// TIA Portal V19 export
DATA_BLOCK "MwFakCalc_PERS"   // DB132
// stored: MemoryReserve 100
   VAR RETAIN
      PersistentValues : "udt_MwFacCalc_Pers";
   END_VAR
BEGIN
   PersistentValues.Data.MaterialPresence := TRUE;
   PersistentValues.Data.Reg[1].ID := 713;
   PersistentValues.Data.Reg[2].ID := 712;
   PersistentValues.Data.Reg[3].ID := 711;
   PersistentValues.Data.Reg[4].ID := 710;
   PersistentValues.Data.Reg[5].ID := 709;
   PersistentValues.Data.Reg[6].ID := 708;
   PersistentValues.Data.Reg[7].ID := 707;
   PersistentValues.Data.Reg[8].ID := 706;
   PersistentValues.Data.Reg[9].ID := 705;
   PersistentValues.Data.Reg[10].ID := 704;
   PersistentValues.Data.Reg[1].FAK := 1.00032760149922;
   PersistentValues.Data.Reg[2].FAK := 1.00025286183891;
   PersistentValues.Data.Reg[3].FAK := 1.00034141784116;
   PersistentValues.Data.Reg[4].FAK := 1.00032858034714;
   PersistentValues.Data.Reg[5].FAK := 1.00027275466515;
   PersistentValues.Data.Reg[6].FAK := 1.00033876404002;
   PersistentValues.Data.Reg[7].FAK := 1.00043144089834;
   PersistentValues.Data.Reg[8].FAK := 1.00027468282716;
   PersistentValues.Data.Reg[9].FAK := 1.0002702312408;
   PersistentValues.Data.Reg[10].FAK := 1.00040598281433;
   PersistentValues.Data.Reg[1].FAK_PS := 1.00033187802923;
   PersistentValues.Data.Reg[2].FAK_PS := 1.0002428384096;
   PersistentValues.Data.Reg[3].FAK_PS := 1.00034713591431;
   PersistentValues.Data.Reg[4].FAK_PS := 1.0003300372471;
   PersistentValues.Data.Reg[5].FAK_PS := 1.00028276221556;
   PersistentValues.Data.Reg[6].FAK_PS := 1.0003416145074;
   PersistentValues.Data.Reg[7].FAK_PS := 1.00041568993821;
   PersistentValues.Data.Reg[8].FAK_PS := 1.00027756475559;
   PersistentValues.Data.Reg[9].FAK_PS := 1.00025879029114;
   PersistentValues.Data.Reg[10].FAK_PS := 1.00039311435194;
   PersistentValues.Data.Reg[1].TP_W_Meas1Reg.ID := 1347;
   PersistentValues.Data.Reg[2].TP_W_Meas1Reg.ID := 1345;
   PersistentValues.Data.Reg[3].TP_W_Meas1Reg.ID := 1343;
   PersistentValues.Data.Reg[4].TP_W_Meas1Reg.ID := 1341;
   PersistentValues.Data.Reg[5].TP_W_Meas1Reg.ID := 1339;
   PersistentValues.Data.Reg[6].TP_W_Meas1Reg.ID := 1337;
   PersistentValues.Data.Reg[7].TP_W_Meas1Reg.ID := 1335;
   PersistentValues.Data.Reg[8].TP_W_Meas1Reg.ID := 1333;
   PersistentValues.Data.Reg[9].TP_W_Meas1Reg.ID := 1331;
   PersistentValues.Data.Reg[10].TP_W_Meas1Reg.ID := 1329;
   PersistentValues.Data.Reg[1].TP_W_Meas1Reg.Position := 900953.878;
   PersistentValues.Data.Reg[2].TP_W_Meas1Reg.Position := 898853.79;
   PersistentValues.Data.Reg[3].TP_W_Meas1Reg.Position := 896756.481;
   PersistentValues.Data.Reg[4].TP_W_Meas1Reg.Position := 895002.073;
   PersistentValues.Data.Reg[5].TP_W_Meas1Reg.Position := 892900.793;
   PersistentValues.Data.Reg[6].TP_W_Meas1Reg.Position := 890799.166;
   PersistentValues.Data.Reg[7].TP_W_Meas1Reg.Position := 888692.332;
   PersistentValues.Data.Reg[8].TP_W_Meas1Reg.Position := 886941.647;
   PersistentValues.Data.Reg[9].TP_W_Meas1Reg.Position := 884838.939;
   PersistentValues.Data.Reg[10].TP_W_Meas1Reg.Position := 882730.285;
   PersistentValues.Data.Reg[1].TP_G_Meas1Reg.ID := 1346;
   PersistentValues.Data.Reg[2].TP_G_Meas1Reg.ID := 1344;
   PersistentValues.Data.Reg[3].TP_G_Meas1Reg.ID := 1342;
   PersistentValues.Data.Reg[4].TP_G_Meas1Reg.ID := 1340;
   PersistentValues.Data.Reg[5].TP_G_Meas1Reg.ID := 1338;
   PersistentValues.Data.Reg[6].TP_G_Meas1Reg.ID := 1336;
   PersistentValues.Data.Reg[7].TP_G_Meas1Reg.ID := 1334;
   PersistentValues.Data.Reg[8].TP_G_Meas1Reg.ID := 1332;
   PersistentValues.Data.Reg[9].TP_G_Meas1Reg.ID := 1330;
   PersistentValues.Data.Reg[10].TP_G_Meas1Reg.ID := 1328;
   PersistentValues.Data.Reg[1].TP_G_Meas1Reg.Position := -650.875;
   PersistentValues.Data.Reg[2].TP_G_Meas1Reg.Position := -651.608;
   PersistentValues.Data.Reg[3].TP_G_Meas1Reg.Position := -652.018;
   PersistentValues.Data.Reg[4].TP_G_Meas1Reg.Position := -651.902;
   PersistentValues.Data.Reg[5].TP_G_Meas1Reg.Position := -652.251;
   PersistentValues.Data.Reg[6].TP_G_Meas1Reg.Position := -651.557;
   PersistentValues.Data.Reg[7].TP_G_Meas1Reg.Position := -651.833;
   PersistentValues.Data.Reg[8].TP_G_Meas1Reg.Position := -650.823;
   PersistentValues.Data.Reg[9].TP_G_Meas1Reg.Position := -651.386;
   PersistentValues.Data.Reg[10].TP_G_Meas1Reg.Position := -652.001;
   PersistentValues.Data.Reg[1].TP_W_Meas2Reg.ID := 1348;
   PersistentValues.Data.Reg[2].TP_W_Meas2Reg.ID := 1346;
   PersistentValues.Data.Reg[3].TP_W_Meas2Reg.ID := 1344;
   PersistentValues.Data.Reg[4].TP_W_Meas2Reg.ID := 1342;
   PersistentValues.Data.Reg[5].TP_W_Meas2Reg.ID := 1340;
   PersistentValues.Data.Reg[6].TP_W_Meas2Reg.ID := 1338;
   PersistentValues.Data.Reg[7].TP_W_Meas2Reg.ID := 1336;
   PersistentValues.Data.Reg[8].TP_W_Meas2Reg.ID := 1334;
   PersistentValues.Data.Reg[9].TP_W_Meas2Reg.ID := 1332;
   PersistentValues.Data.Reg[10].TP_W_Meas2Reg.ID := 1330;
   PersistentValues.Data.Reg[1].TP_W_Meas2Reg.Position := 901652.898;
   PersistentValues.Data.Reg[2].TP_W_Meas2Reg.Position := 899553.777;
   PersistentValues.Data.Reg[3].TP_W_Meas2Reg.Position := 897456.503;
   PersistentValues.Data.Reg[4].TP_W_Meas2Reg.Position := 895702.054;
   PersistentValues.Data.Reg[5].TP_W_Meas2Reg.Position := 893601.056;
   PersistentValues.Data.Reg[6].TP_W_Meas2Reg.Position := 891498.768;
   PersistentValues.Data.Reg[7].TP_W_Meas2Reg.Position := 889392.312;
   PersistentValues.Data.Reg[8].TP_W_Meas2Reg.Position := 887640.635;
   PersistentValues.Data.Reg[9].TP_W_Meas2Reg.Position := 885538.34;
   PersistentValues.Data.Reg[10].TP_W_Meas2Reg.Position := 883429.822;
   PersistentValues.Data.Reg[1].TP_G_Meas2Reg.ID := 1347;
   PersistentValues.Data.Reg[2].TP_G_Meas2Reg.ID := 1345;
   PersistentValues.Data.Reg[3].TP_G_Meas2Reg.ID := 1343;
   PersistentValues.Data.Reg[4].TP_G_Meas2Reg.ID := 1341;
   PersistentValues.Data.Reg[5].TP_G_Meas2Reg.ID := 1339;
   PersistentValues.Data.Reg[6].TP_G_Meas2Reg.ID := 1337;
   PersistentValues.Data.Reg[7].TP_G_Meas2Reg.ID := 1335;
   PersistentValues.Data.Reg[8].TP_G_Meas2Reg.ID := 1333;
   PersistentValues.Data.Reg[9].TP_G_Meas2Reg.ID := 1331;
   PersistentValues.Data.Reg[10].TP_G_Meas2Reg.ID := 1329;
   PersistentValues.Data.Reg[1].TP_G_Meas2Reg.Position := 48.374;
   PersistentValues.Data.Reg[2].TP_G_Meas2Reg.Position := 48.556;
   PersistentValues.Data.Reg[3].TP_G_Meas2Reg.Position := 48.243;
   PersistentValues.Data.Reg[4].TP_G_Meas2Reg.Position := 48.309;
   PersistentValues.Data.Reg[5].TP_G_Meas2Reg.Position := 48.203;
   PersistentValues.Data.Reg[6].TP_G_Meas2Reg.Position := 48.282;
   PersistentValues.Data.Reg[7].TP_G_Meas2Reg.Position := 48.449;
   PersistentValues.Data.Reg[8].TP_G_Meas2Reg.Position := 48.357;
   PersistentValues.Data.Reg[9].TP_G_Meas2Reg.Position := 48.204;
   PersistentValues.Data.Reg[10].TP_G_Meas2Reg.Position := 47.82;
   PersistentValues.Data.Reg[1].PS_W_Meas1Reg.ID := 217;
   PersistentValues.Data.Reg[2].PS_W_Meas1Reg.ID := 215;
   PersistentValues.Data.Reg[3].PS_W_Meas1Reg.ID := 213;
   PersistentValues.Data.Reg[4].PS_W_Meas1Reg.ID := 211;
   PersistentValues.Data.Reg[5].PS_W_Meas1Reg.ID := 209;
   PersistentValues.Data.Reg[6].PS_W_Meas1Reg.ID := 207;
   PersistentValues.Data.Reg[7].PS_W_Meas1Reg.ID := 205;
   PersistentValues.Data.Reg[8].PS_W_Meas1Reg.ID := 203;
   PersistentValues.Data.Reg[9].PS_W_Meas1Reg.ID := 201;
   PersistentValues.Data.Reg[10].PS_W_Meas1Reg.ID := 199;
   PersistentValues.Data.Reg[1].PS_W_Meas1Reg.Position := 900953.482;
   PersistentValues.Data.Reg[2].PS_W_Meas1Reg.Position := 898853.373;
   PersistentValues.Data.Reg[3].PS_W_Meas1Reg.Position := 896756.134;
   PersistentValues.Data.Reg[4].PS_W_Meas1Reg.Position := 895001.723;
   PersistentValues.Data.Reg[5].PS_W_Meas1Reg.Position := 892900.467;
   PersistentValues.Data.Reg[6].PS_W_Meas1Reg.Position := 890798.798;
   PersistentValues.Data.Reg[7].PS_W_Meas1Reg.Position := 888691.934;
   PersistentValues.Data.Reg[8].PS_W_Meas1Reg.Position := 886941.298;
   PersistentValues.Data.Reg[9].PS_W_Meas1Reg.Position := 884838.507;
   PersistentValues.Data.Reg[10].PS_W_Meas1Reg.Position := 882729.938;
   PersistentValues.Data.Reg[1].PS_G_Meas1Reg.ID := 217;
   PersistentValues.Data.Reg[2].PS_G_Meas1Reg.ID := 215;
   PersistentValues.Data.Reg[3].PS_G_Meas1Reg.ID := 213;
   PersistentValues.Data.Reg[4].PS_G_Meas1Reg.ID := 211;
   PersistentValues.Data.Reg[5].PS_G_Meas1Reg.ID := 209;
   PersistentValues.Data.Reg[6].PS_G_Meas1Reg.ID := 207;
   PersistentValues.Data.Reg[7].PS_G_Meas1Reg.ID := 205;
   PersistentValues.Data.Reg[8].PS_G_Meas1Reg.ID := 203;
   PersistentValues.Data.Reg[9].PS_G_Meas1Reg.ID := 201;
   PersistentValues.Data.Reg[10].PS_G_Meas1Reg.ID := 199;
   PersistentValues.Data.Reg[1].PS_G_Meas1Reg.Position := -651.256;
   PersistentValues.Data.Reg[2].PS_G_Meas1Reg.Position := -652.0;
   PersistentValues.Data.Reg[3].PS_G_Meas1Reg.Position := -652.349;
   PersistentValues.Data.Reg[4].PS_G_Meas1Reg.Position := -652.229;
   PersistentValues.Data.Reg[5].PS_G_Meas1Reg.Position := -652.553;
   PersistentValues.Data.Reg[6].PS_G_Meas1Reg.Position := -651.902;
   PersistentValues.Data.Reg[7].PS_G_Meas1Reg.Position := -652.202;
   PersistentValues.Data.Reg[8].PS_G_Meas1Reg.Position := -651.153;
   PersistentValues.Data.Reg[9].PS_G_Meas1Reg.Position := -651.791;
   PersistentValues.Data.Reg[10].PS_G_Meas1Reg.Position := -652.328;
   PersistentValues.Data.Reg[1].PS_W_Meas2Reg.ID := 218;
   PersistentValues.Data.Reg[2].PS_W_Meas2Reg.ID := 216;
   PersistentValues.Data.Reg[3].PS_W_Meas2Reg.ID := 214;
   PersistentValues.Data.Reg[4].PS_W_Meas2Reg.ID := 212;
   PersistentValues.Data.Reg[5].PS_W_Meas2Reg.ID := 210;
   PersistentValues.Data.Reg[6].PS_W_Meas2Reg.ID := 208;
   PersistentValues.Data.Reg[7].PS_W_Meas2Reg.ID := 206;
   PersistentValues.Data.Reg[8].PS_W_Meas2Reg.ID := 204;
   PersistentValues.Data.Reg[9].PS_W_Meas2Reg.ID := 202;
   PersistentValues.Data.Reg[10].PS_W_Meas2Reg.ID := 200;
   PersistentValues.Data.Reg[1].PS_W_Meas2Reg.Position := 901652.534;
   PersistentValues.Data.Reg[2].PS_W_Meas2Reg.Position := 899553.427;
   PersistentValues.Data.Reg[3].PS_W_Meas2Reg.Position := 897456.148;
   PersistentValues.Data.Reg[4].PS_W_Meas2Reg.Position := 895701.644;
   PersistentValues.Data.Reg[5].PS_W_Meas2Reg.Position := 893600.702;
   PersistentValues.Data.Reg[6].PS_W_Meas2Reg.Position := 891498.417;
   PersistentValues.Data.Reg[7].PS_W_Meas2Reg.Position := 889391.975;
   PersistentValues.Data.Reg[8].PS_W_Meas2Reg.Position := 887640.234;
   PersistentValues.Data.Reg[9].PS_W_Meas2Reg.Position := 885537.915;
   PersistentValues.Data.Reg[10].PS_W_Meas2Reg.Position := 883429.48;
   PersistentValues.Data.Reg[1].PS_G_Meas2Reg.ID := 218;
   PersistentValues.Data.Reg[2].PS_G_Meas2Reg.ID := 216;
   PersistentValues.Data.Reg[3].PS_G_Meas2Reg.ID := 214;
   PersistentValues.Data.Reg[4].PS_G_Meas2Reg.ID := 212;
   PersistentValues.Data.Reg[5].PS_G_Meas2Reg.ID := 210;
   PersistentValues.Data.Reg[6].PS_G_Meas2Reg.ID := 208;
   PersistentValues.Data.Reg[7].PS_G_Meas2Reg.ID := 206;
   PersistentValues.Data.Reg[8].PS_G_Meas2Reg.ID := 204;
   PersistentValues.Data.Reg[9].PS_G_Meas2Reg.ID := 202;
   PersistentValues.Data.Reg[10].PS_G_Meas2Reg.ID := 200;
   PersistentValues.Data.Reg[1].PS_G_Meas2Reg.Position := 48.028;
   PersistentValues.Data.Reg[2].PS_G_Meas2Reg.Position := 48.224;
   PersistentValues.Data.Reg[3].PS_G_Meas2Reg.Position := 47.908;
   PersistentValues.Data.Reg[4].PS_G_Meas2Reg.Position := 47.923;
   PersistentValues.Data.Reg[5].PS_G_Meas2Reg.Position := 47.88;
   PersistentValues.Data.Reg[6].PS_G_Meas2Reg.Position := 47.956;
   PersistentValues.Data.Reg[7].PS_G_Meas2Reg.Position := 48.13;
   PersistentValues.Data.Reg[8].PS_G_Meas2Reg.Position := 47.977;
   PersistentValues.Data.Reg[9].PS_G_Meas2Reg.Position := 47.798;
   PersistentValues.Data.Reg[10].PS_G_Meas2Reg.Position := 47.489;
   PersistentValues.Data.RegItemsValid := 10;
   PersistentValues.Data.RegID := 714;
   PersistentValues.Data.GripperMeasID := 1347;
   PersistentValues.Data.WheelMeasID := 1348;
   PersistentValues.Data.AverageFAK := 1.00032443180122;
   PersistentValues.Par.WorkMode := 1;
   PersistentValues.Par.Gripper_Meas1_PosStart := 200.0;
   PersistentValues.Par.Gripper_Meas1_DonePosLim := 250.0;
   PersistentValues.Par.Gripper_Meas2_PosStart := 700.0;
   PersistentValues.Par.Gripper_Meas2_DonePosLim := 750.0;
   PersistentValues.Par.PushAx.Man.VelBwd := 15000.0;
   PersistentValues.Par.PushAx.Man.VelFwdHigh := 15000.0;
   PersistentValues.Par.PushAx.Man.VelFwdLow := 2000.0;
   PersistentValues.Par.PushAx.Man.Acc := 1000.0;
   PersistentValues.Par.PushAx.Man.Dec := 1000.0;
   PersistentValues.Par.PushAx.Man.DelayChangeVel := T#1MS;
   PersistentValues.Par.PushAx_Aut_VelHigh := 18000.0;
   PersistentValues.Par.PushAx_Aut_VelLow := 4000.0;
   PersistentValues.Par.PushAx_Aut_Acc := 1000.0;
   PersistentValues.Par.PushAx_Aut_Dec := 1000.0;
END_DATA_BLOCK
